// TIA Portal V19 export
DATA_BLOCK "NetworkSwitchFaceplate_DB"   // DB32
// stored: InstanceOfName NetworkSwitchFaceplate, InstanceOfType FB
"NetworkSwitchFaceplate"
   // VAR_INPUT
   //    Index : Int;
   // END_VAR
   // VAR_OUTPUT
   //    PeerName { ExternalAccessible := 'False'; ExternalVisible := 'False'; ExternalWritable := 'False'} : String;
   // END_VAR
   // VAR_IN_OUT
   //    Port : "NetworkSwitchHMI";
   // END_VAR
BEGIN
END_DATA_BLOCK
